PROGRAM MAIN
VAR
	bPut: BOOL;
	fbHttpClient: FB_IotHttpClient := (sHostName:= '192.168.1.99',bKeepAlive := TRUE, tConnectionTimeout:=T#10S);
	fbPut: FB_HttpPut;
	bBlinkingMode: BOOL;
	fbTimer: ton := (pt:=T#500MS);
	nColor: UINT;
END_VAR

IF NOT fbHttpClient.bConfigured THEN
	fbHttpClient.nHostPort := 80;
	fbHttpClient.stTLS.bNoServerCertCheck:= TRUE;
END_IF

IF fbHttpClient.bConfigured THEN
	fbPut(bSend := bPut, fbClient:= fbHttpClient, nColor:= nColor);
END_IF

IF bBlinkingMode THEN
	fbTimer(in:= NOT fbTimer.Q);
	IF fbTimer.Q THEN
		nColor:=nColor+5000;
        IF nColor=65000 THEN
            nColor:=0;
        END_IF
		IF bPut THEN
			bPut:= FALSE;
		ELSE
			bPut:= TRUE;
		END_IF
	END_IF
END_IF

fbHttpClient.Execute();

END_PROGRAM

(* stored: Version 1.1.0.1, ProductVersion 3.1.4024.4
   POU MAIN: Id {e7f8665c-0059-4525-8a94-e2650ae2c275}, SpecialFunc None *)
